FUNCTION TIMESTAMP_NS (* creates default a Unix-Epoch-Timestamp in nanoseconds use other start dates for other timestamp types *)
  PACKAGE eclipse4diac::utils::timing;
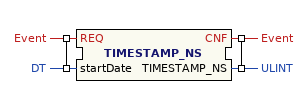
  EVENT_INPUT
    REQ WITH startDate; (* request to create a timestamp *)
  END_EVENT
  EVENT_OUTPUT
    CNF WITH TIMESTAMP_NS; (* confirms the creation of a timestamp *)
  END_EVENT
  VAR_INPUT
    startDate : DT := DT#1970-01-01-00:00:00; (* the start date used to calculate different timestamp types *)
  END_VAR
  VAR_OUTPUT
    TIMESTAMP_NS : ULINT; (* the new timestamp in nanoseconds, default Unix-Epoch *)
  END_VAR
  BODY IN ST:
FUNCTION TIMESTAMP_NS : ULINT
VAR_INPUT
	startDate : DT := DT#1970-01-01-00:00:00;
END_VAR
TIMESTAMP_NS := TIME_IN_NS_TO_ULINT(NOW() - startDate);
END_FUNCTION
  END_BODY
END_FUNCTION
